(* PLC project rien, Dassault Systèmes ControlBuild 2024x Refresh1 *)
(* stored: creationDateTime 2024-03-20T17:34:47-01:00 *)

PROGRAM aaaaa
  VAR_INPUT
    s : BOOL := false;
    s2 : BOOL := false;
  END_VAR

(* FBD diagram, written out as Structured Text *)
END_PROGRAM

PROGRAM zozo.rien
  VAR_INPUT
    s : BOOL := false;
    s2 : BOOL := false;
  END_VAR

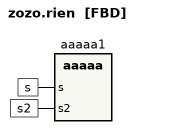
(* FBD diagram, written out as Structured Text *)
aaaaa1(s := s, s2 := s2);
END_PROGRAM
